Staubli VAL3: cycleStatus.pjx

--- cycleStatus.pjx ---
Parameters version=s7.4 stackSize=5000 millimeterUnit=true
Data file=cycleStatus.dtx

--- cycleStatus.dtx ---
public bool bAllInHome
public bool bAxis13Running
public bool bCycle
public bool bDebug
public bool bFinishCycle
public bool bManualMode = true
public bool bMoveStopped
public bool bPause
public bool bPcStartCycle
public bool bPcStopCycle
public bool bQuit
public bool bRemoteMode
public bool bRtCalibrated = true
public bool bRtRbtEstop
public bool bRtRbtInHome
public bool bRtRbtReady
public bool bToStop = true
public bool bWorkingMode = true
public num nProcedure
public num nToSuperV = -1
public num nWorkingMode = 1
public num nWorkingStatus = 6
